INTERFACE I_GraphFactory

METHOD PUBLIC Accept
VAR_INPUT
	Visitor : I_GraphFactoryVisitor;
END_VAR
END_METHOD

METHOD PUBLIC Create : I_Graph
VAR_INPUT
END_VAR
END_METHOD

METHOD PUBLIC GetNodePrototypes : I_NodePrototypes
VAR_INPUT
END_VAR
END_METHOD

METHOD PUBLIC InstallNodePack
VAR_INPUT
	NodePack : I_NodePack;
END_VAR
END_METHOD

METHOD PUBLIC RegisterNodeByType
VAR_INPUT
	NodeType : T_MAXSTRING;
	NodePrototype : I_NodePrototype;	
END_VAR
END_METHOD

END_INTERFACE

(* stored: Version 1.1.0.1, ProductVersion 3.1.4024.12
   Itf I_GraphFactory: Id {baf0ca6a-df37-0eff-28cb-e8832601c45e}
   Method Accept: Id {d6b0227b-c6be-0b92-292f-1c6818ca100e}
   Method Create: Id {1854d952-a565-0180-3eca-962fe7a561ac}
   Method GetNodePrototypes: Id {fe605af4-4f06-48e6-8672-71b3b58eab8c}
   Method InstallNodePack: Id {a1b01422-7833-00b5-0b04-6d2dd72028e7}
   Method RegisterNodeByType: Id {3f521954-a6e6-0df9-3dcf-fc038d75e218} *)
